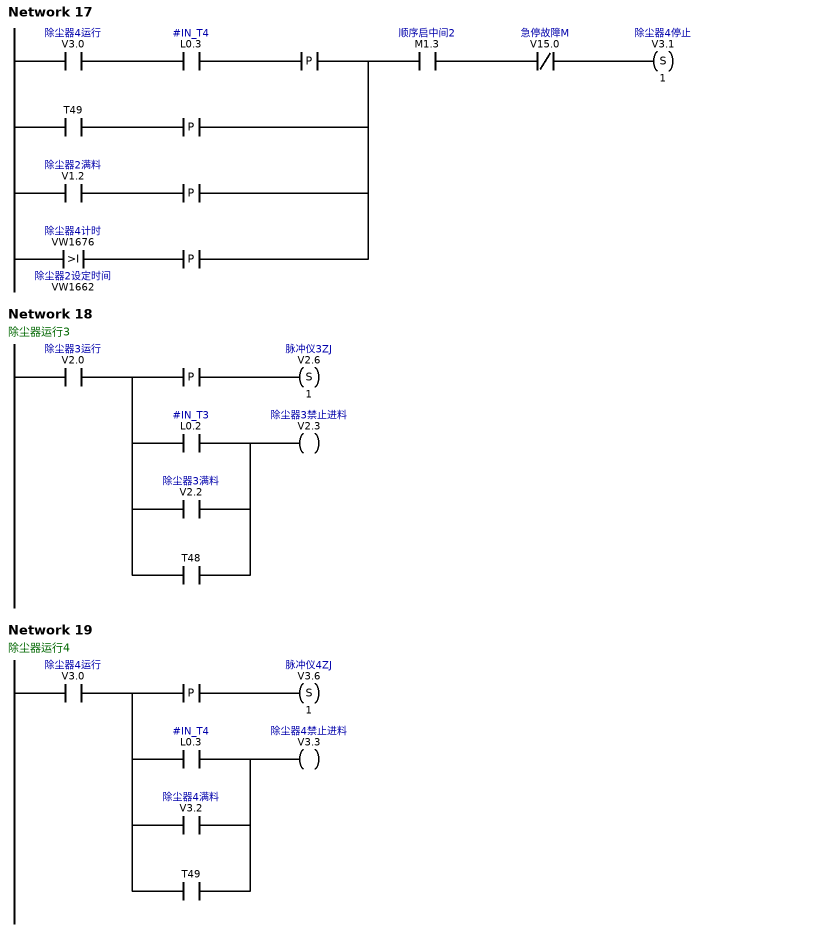
[picture p96: SBR29 networks 17-19]
Network 17
LD     除尘器4运行:V3.0
A      #IN_T4:L0.3
EU
LD     T49
EU
OLD
LD     除尘器2满料:V1.2
EU
OLD
LDW>   除尘器4计时:VW1676, 除尘器2设定时间:VW1662
EU
OLD
A      顺序启中间2:M1.3
AN     急停故障M:V15.0
S      除尘器4停止:V3.1, 1
Network 18
// 除尘器运行3
LD     除尘器3运行:V2.0
LPS
EU
S      脉冲仪3ZJ:V2.6, 1
LPP
LD     #IN_T3:L0.2
O      除尘器3满料:V2.2
O      T48
ALD
=      除尘器3禁止进料:V2.3
Network 19
// 除尘器运行4
LD     除尘器4运行:V3.0
LPS
EU
S      脉冲仪4ZJ:V3.6, 1
LPP
LD     #IN_T4:L0.3
O      除尘器4满料:V3.2
O      T49
ALD
=      除尘器4禁止进料:V3.3
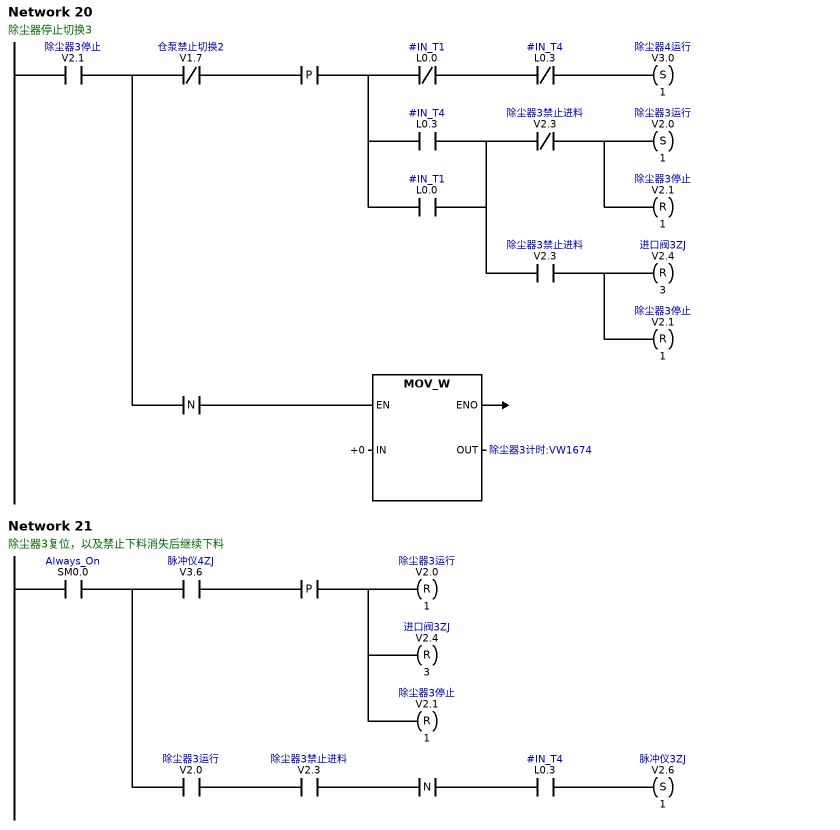
Network 20
// 除尘器停止切换3
LD     除尘器3停止:V2.1
LPS
AN     仓泵禁止切换2:V1.7
EU
LPS
AN     #IN_T1:L0.0
AN     #IN_T4:L0.3
S      除尘器4运行:V3.0, 1
LPP
LD     #IN_T4:L0.3
O      #IN_T1:L0.0
ALD
LPS
AN     除尘器3禁止进料:V2.3
S      除尘器3运行:V2.0, 1
R      除尘器3停止:V2.1, 1
LPP
A      除尘器3禁止进料:V2.3
R      进口阀3ZJ:V2.4, 3
R      除尘器3停止:V2.1, 1
LPP
ED
MOVW   +0, 除尘器3计时:VW1674
Network 21
// 除尘器3复位，以及禁止下料消失后继续下料
LD     Always_On:SM0.0
LPS
A      脉冲仪4ZJ:V3.6
EU
R      除尘器3运行:V2.0, 1
R      进口阀3ZJ:V2.4, 3
R      除尘器3停止:V2.1, 1
LPP
A      除尘器3运行:V2.0
A      除尘器3禁止进料:V2.3
ED
A      #IN_T4:L0.3
S      脉冲仪3ZJ:V2.6, 1
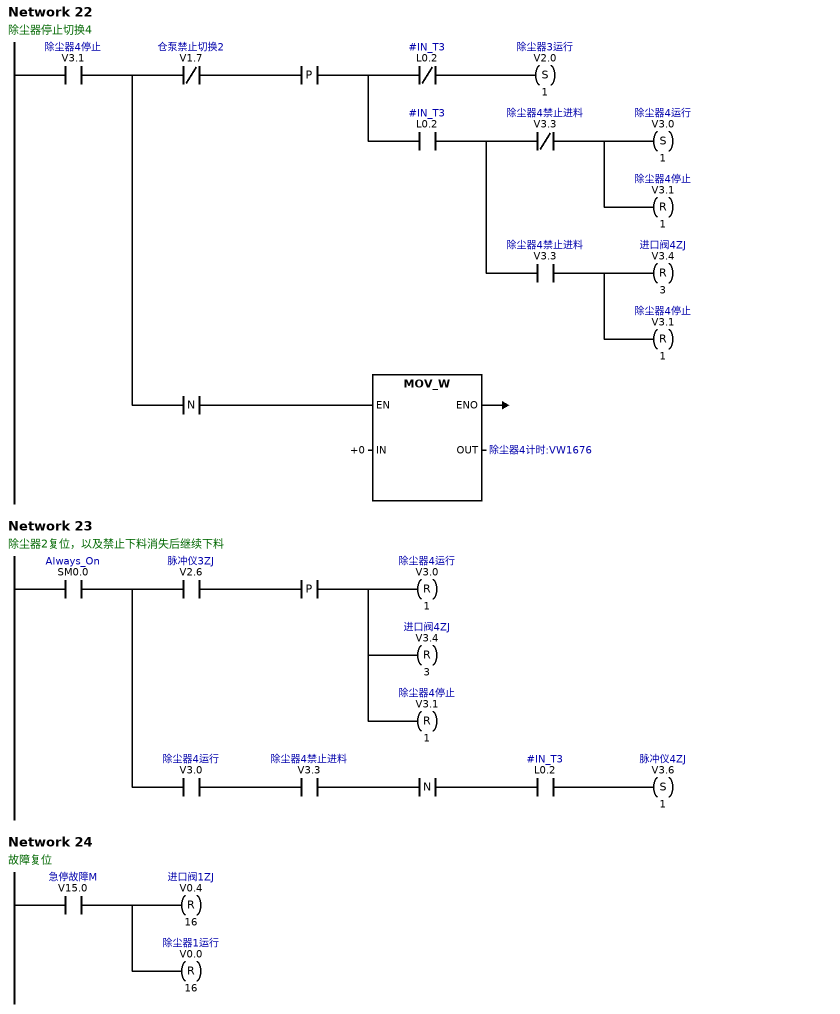
Network 22
// 除尘器停止切换4
LD     除尘器4停止:V3.1
LPS
AN     仓泵禁止切换2:V1.7
EU
LPS
AN     #IN_T3:L0.2
S      除尘器3运行:V2.0, 1
LPP
A      #IN_T3:L0.2
LPS
AN     除尘器4禁止进料:V3.3
S      除尘器4运行:V3.0, 1
R      除尘器4停止:V3.1, 1
LPP
A      除尘器4禁止进料:V3.3
R      进口阀4ZJ:V3.4, 3
R      除尘器4停止:V3.1, 1
LPP
ED
MOVW   +0, 除尘器4计时:VW1676
Network 23
// 除尘器2复位，以及禁止下料消失后继续下料
LD     Always_On:SM0.0
LPS
A      脉冲仪3ZJ:V2.6
EU
R      除尘器4运行:V3.0, 1
R      进口阀4ZJ:V3.4, 3
R      除尘器4停止:V3.1, 1
LPP
A      除尘器4运行:V3.0
A      除尘器4禁止进料:V3.3
ED
A      #IN_T3:L0.2
S      脉冲仪4ZJ:V3.6, 1
Network 24
// 故障复位
LD     急停故障M:V15.0
R      进口阀1ZJ:V0.4, 16
R      除尘器1运行:V0.0, 16
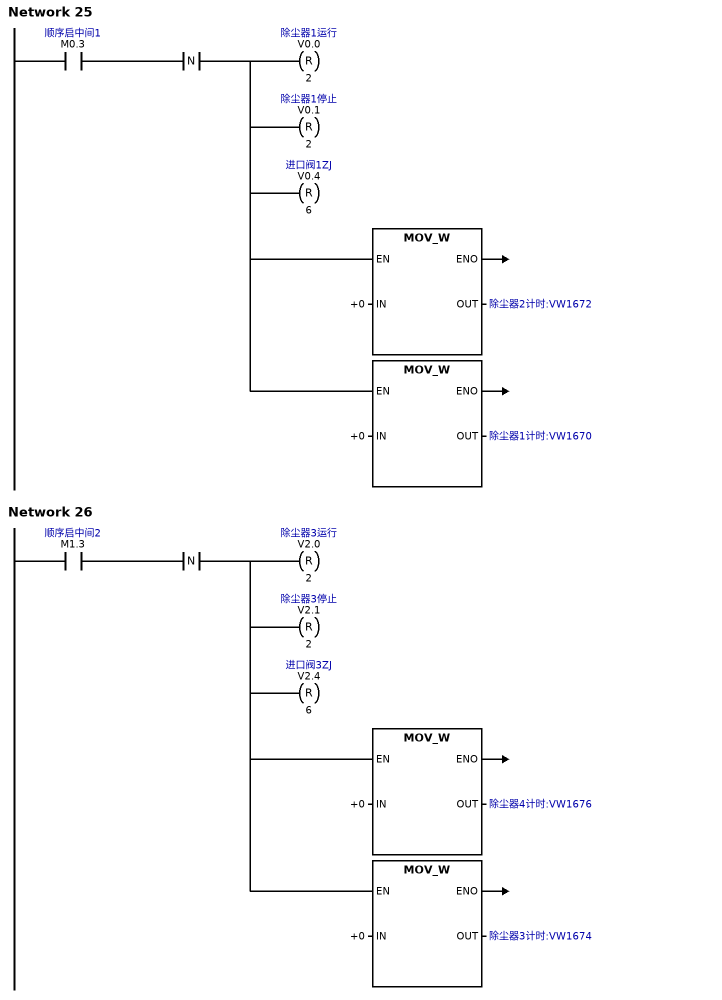
Network 25
LD     顺序启中间1:M0.3
ED
R      除尘器1运行:V0.0, 2
R      除尘器1停止:V0.1, 2
R      进口阀1ZJ:V0.4, 6
MOVW   +0, 除尘器2计时:VW1672
MOVW   +0, 除尘器1计时:VW1670
Network 26
LD     顺序启中间2:M1.3
ED
R      除尘器3运行:V2.0, 2
R      除尘器3停止:V2.1, 2
R      进口阀3ZJ:V2.4, 6
MOVW   +0, 除尘器4计时:VW1676
MOVW   +0, 除尘器3计时:VW1674
END_SUBROUTINE_BLOCK

SUBROUTINE_BLOCK MODBUS_XMZ:SBR50
TITLE=
BEGIN
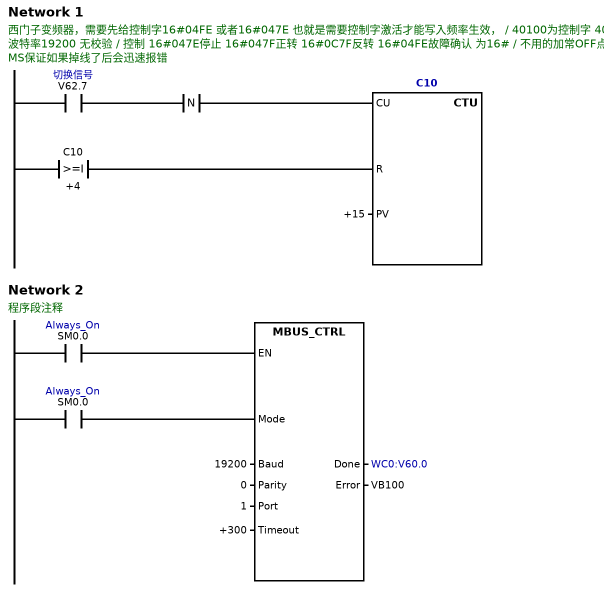
Network 1
// 西门子变频器，需要先给控制字16#04FE 或者16#047E 也就是需要控制字激活才能写入频率生效，
// 40100为控制字 40101为频率 0~16384=0~100% 
// 40342为频率 40345为电流 小数点通常2位  1  4
// 波特率19200 无校验
// 控制 16#047E停止 16#047F正转 16#0C7F反转 16#04FE故障确认 为16#
// 不用的加常OFF点屏蔽避免出错 也就是C10>=4时，=5的必须加常闭的sm0.0 超时300 MS保证如果掉线了后会迅速报错
LD     切换信号:V62.7
ED
LDW>=  C10, +4
CTU    C10, +15
Network 2
// 程序段注释
LD     Always_On:SM0.0
=      L60.0
LD     Always_On:SM0.0
=      L63.7
LD     L60.0
CALL   MBUS_CTRL:SBR2, L63.7, 19200, 0, 1, +300, WC0:V60.0, VB100
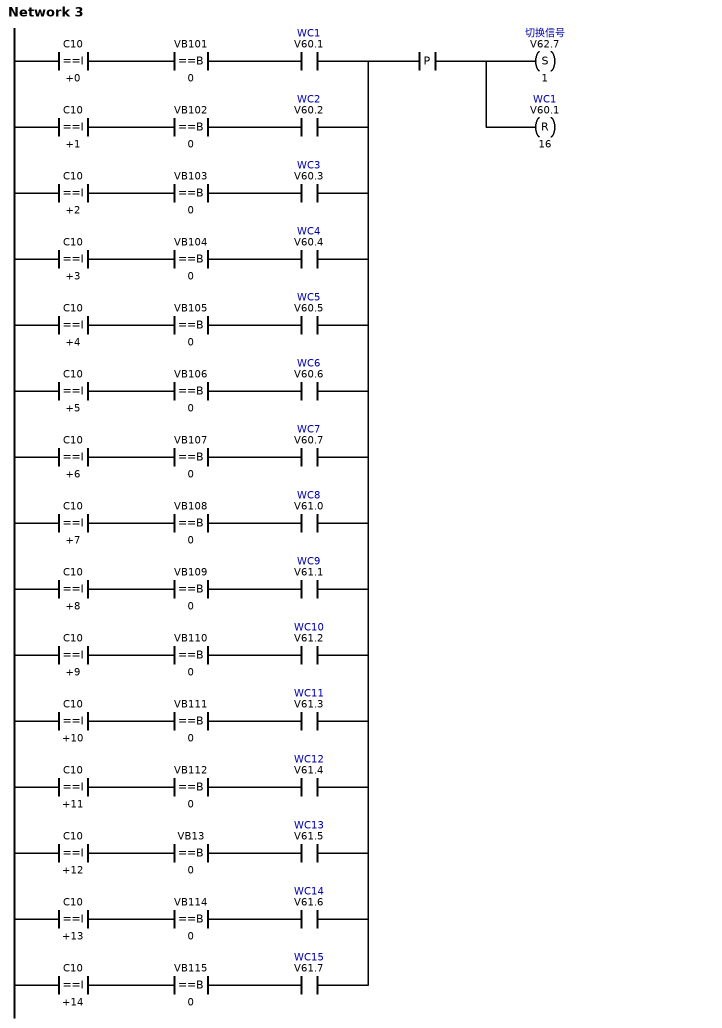
Network 3
LDW=   C10, +0
AB=    VB101, 0
A      WC1:V60.1
LDW=   C10, +1
AB=    VB102, 0
A      WC2:V60.2
OLD
LDW=   C10, +2
AB=    VB103, 0
A      WC3:V60.3
OLD
LDW=   C10, +3
AB=    VB104, 0
A      WC4:V60.4
OLD
LDW=   C10, +4
AB=    VB105, 0
A      WC5:V60.5
OLD
LDW=   C10, +5
AB=    VB106, 0
A      WC6:V60.6
OLD
LDW=   C10, +6
AB=    VB107, 0
A      WC7:V60.7
OLD
LDW=   C10, +7
AB=    VB108, 0
A      WC8:V61.0
OLD
LDW=   C10, +8
AB=    VB109, 0
A      WC9:V61.1
OLD
LDW=   C10, +9
AB=    VB110, 0
A      WC10:V61.2
OLD
LDW=   C10, +10
AB=    VB111, 0
A      WC11:V61.3
OLD
LDW=   C10, +11
AB=    VB112, 0
A      WC12:V61.4
OLD
LDW=   C10, +12
AB=    VB13, 0
A      WC13:V61.5
OLD
LDW=   C10, +13
AB=    VB114, 0
A      WC14:V61.6
OLD
LDW=   C10, +14
AB=    VB115, 0
A      WC15:V61.7
OLD
EU
S      切换信号:V62.7, 1
R      WC1:V60.1, 16
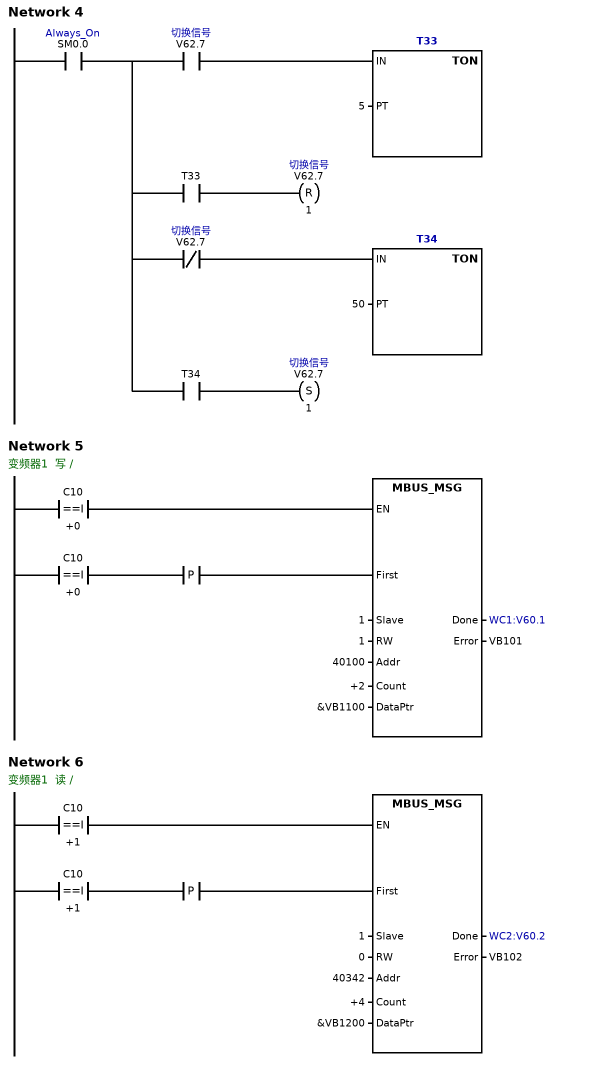
Network 4
LD     Always_On:SM0.0
LPS
A      切换信号:V62.7
TON    T33, 5
LRD
A      T33
R      切换信号:V62.7, 1
LRD
AN     切换信号:V62.7
TON    T34, 50
LPP
A      T34
S      切换信号:V62.7, 1
Network 5
// 变频器1  写
// 
LDW=   C10, +0
=      L60.0
LDW=   C10, +0
EU
=      L63.7
LD     L60.0
CALL   MBUS_MSG:SBR3, L63.7, 1, 1, 40100, +2, &VB1100, WC1:V60.1, VB101
Network 6
// 变频器1  读
// 
LDW=   C10, +1
=      L60.0
LDW=   C10, +1
EU
=      L63.7
LD     L60.0
CALL   MBUS_MSG:SBR3, L63.7, 1, 0, 40342, +4, &VB1200, WC2:V60.2, VB102
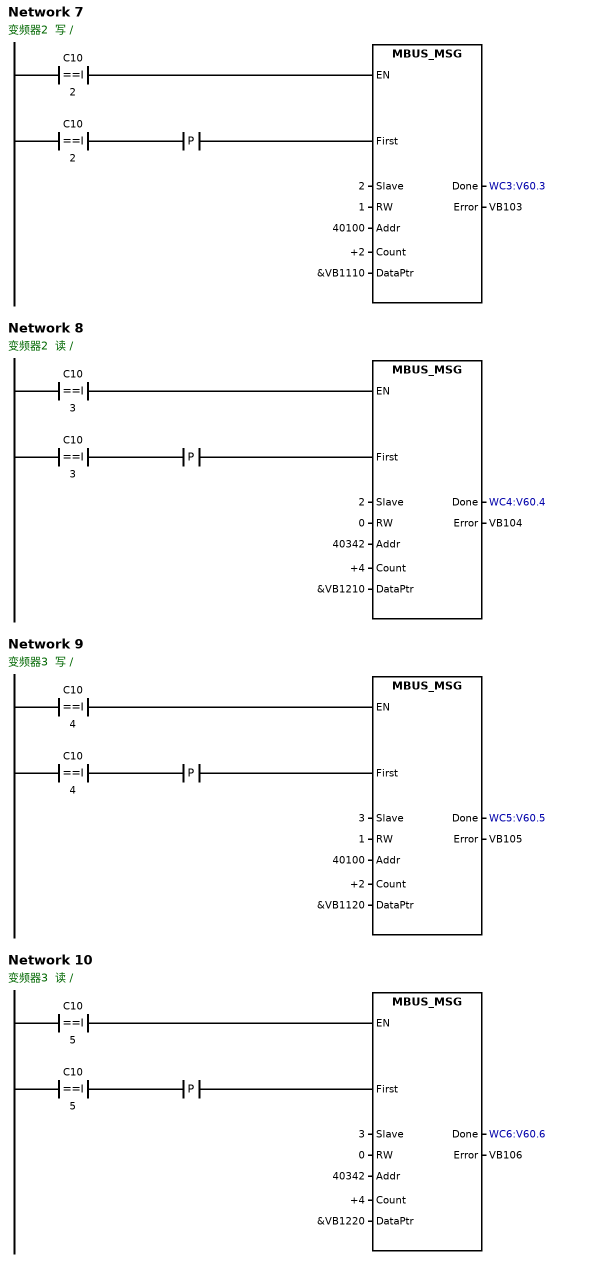
Network 7
// 变频器2  写
// 
LDW=   C10, 2
=      L60.0
LDW=   C10, 2
EU
=      L63.7
LD     L60.0
CALL   MBUS_MSG:SBR3, L63.7, 2, 1, 40100, +2, &VB1110, WC3:V60.3, VB103
Network 8
// 变频器2  读
// 
LDW=   C10, 3
=      L60.0
LDW=   C10, 3
EU
=      L63.7
LD     L60.0
CALL   MBUS_MSG:SBR3, L63.7, 2, 0, 40342, +4, &VB1210, WC4:V60.4, VB104
Network 9
// 变频器3  写
// 
LDW=   C10, 4
=      L60.0
LDW=   C10, 4
EU
=      L63.7
LD     L60.0
CALL   MBUS_MSG:SBR3, L63.7, 3, 1, 40100, +2, &VB1120, WC5:V60.5, VB105
Network 10
// 变频器3  读
// 
LDW=   C10, 5
=      L60.0
LDW=   C10, 5
EU
=      L63.7
LD     L60.0
CALL   MBUS_MSG:SBR3, L63.7, 3, 0, 40342, +4, &VB1220, WC6:V60.6, VB106
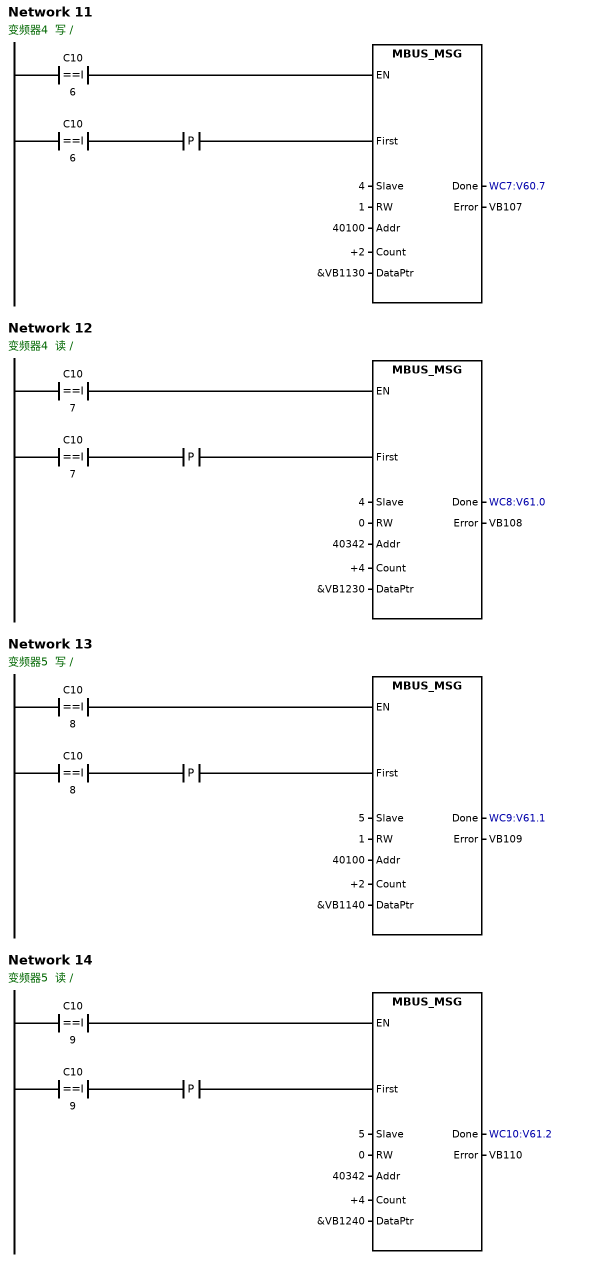
Network 11
// 变频器4  写
// 
LDW=   C10, 6
=      L60.0
LDW=   C10, 6
EU
=      L63.7
LD     L60.0
CALL   MBUS_MSG:SBR3, L63.7, 4, 1, 40100, +2, &VB1130, WC7:V60.7, VB107
Network 12
// 变频器4  读
// 
LDW=   C10, 7
=      L60.0
LDW=   C10, 7
EU
=      L63.7
LD     L60.0
CALL   MBUS_MSG:SBR3, L63.7, 4, 0, 40342, +4, &VB1230, WC8:V61.0, VB108
Network 13
// 变频器5  写
// 
LDW=   C10, 8
=      L60.0
LDW=   C10, 8
EU
=      L63.7
LD     L60.0
CALL   MBUS_MSG:SBR3, L63.7, 5, 1, 40100, +2, &VB1140, WC9:V61.1, VB109
Network 14
// 变频器5  读
// 
LDW=   C10, 9
=      L60.0
LDW=   C10, 9
EU
=      L63.7
LD     L60.0
CALL   MBUS_MSG:SBR3, L63.7, 5, 0, 40342, +4, &VB1240, WC10:V61.2, VB110
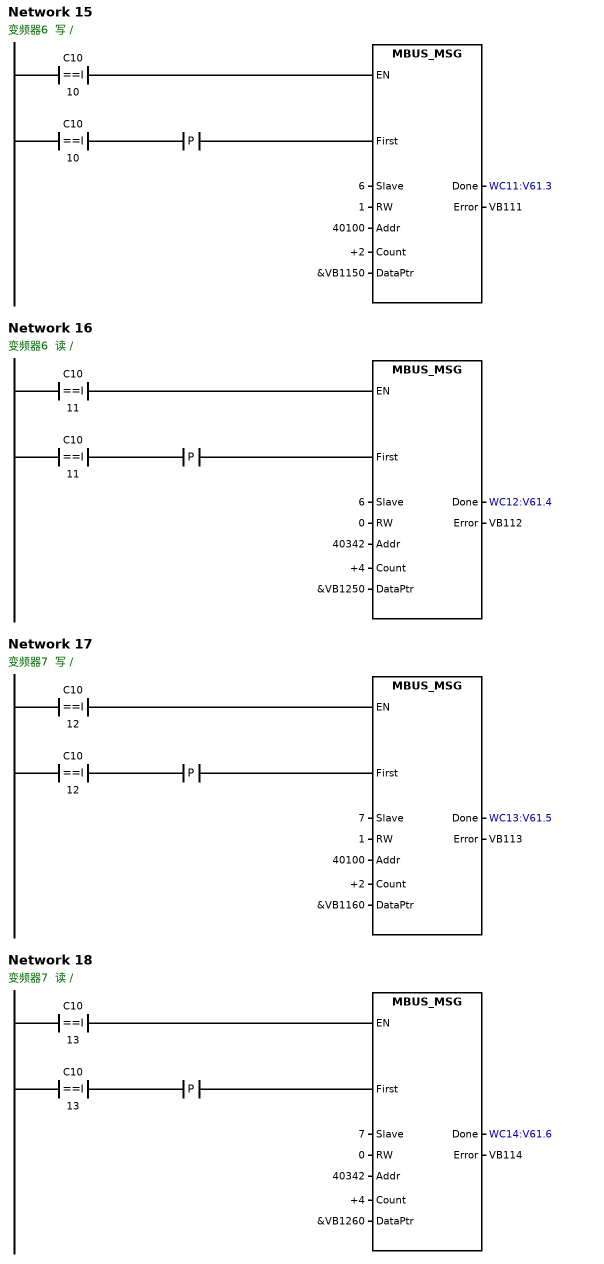
Network 15
// 变频器6  写
// 
LDW=   C10, 10
=      L60.0
LDW=   C10, 10
EU
=      L63.7
LD     L60.0
CALL   MBUS_MSG:SBR3, L63.7, 6, 1, 40100, +2, &VB1150, WC11:V61.3, VB111
Network 16
// 变频器6  读
// 
LDW=   C10, 11
=      L60.0
LDW=   C10, 11
EU
=      L63.7
LD     L60.0
CALL   MBUS_MSG:SBR3, L63.7, 6, 0, 40342, +4, &VB1250, WC12:V61.4, VB112
Network 17
// 变频器7  写
// 
LDW=   C10, 12
=      L60.0
LDW=   C10, 12
EU
=      L63.7
LD     L60.0
CALL   MBUS_MSG:SBR3, L63.7, 7, 1, 40100, +2, &VB1160, WC13:V61.5, VB113
Network 18
// 变频器7  读
// 
LDW=   C10, 13
=      L60.0
LDW=   C10, 13
EU
=      L63.7
LD     L60.0
CALL   MBUS_MSG:SBR3, L63.7, 7, 0, 40342, +4, &VB1260, WC14:V61.6, VB114
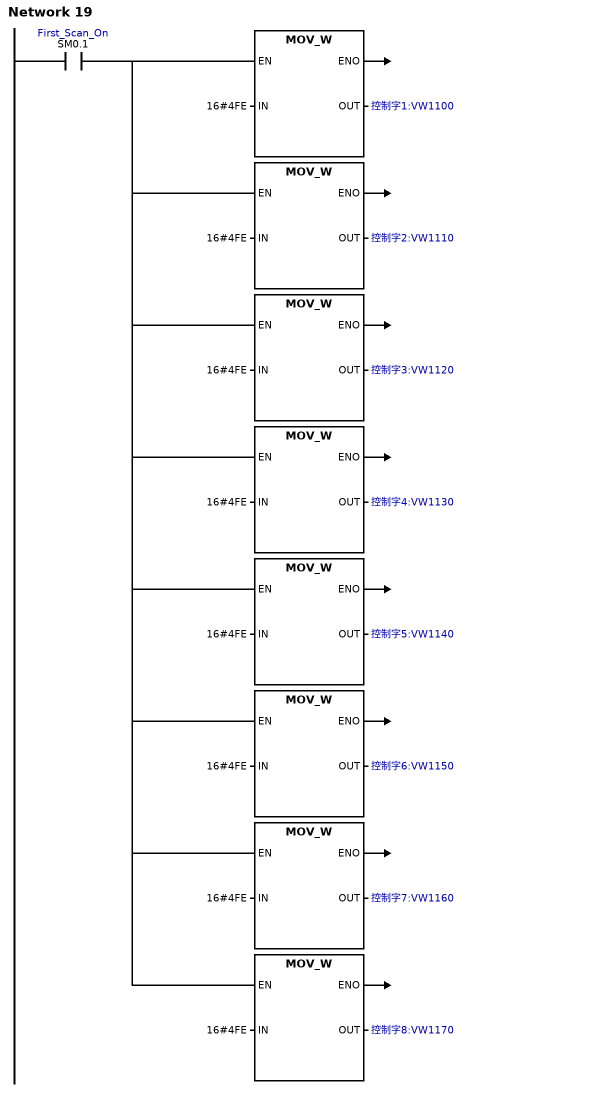
Network 19
LD     First_Scan_On:SM0.1
MOVW   16#4FE, 控制字1:VW1100
MOVW   16#4FE, 控制字2:VW1110
MOVW   16#4FE, 控制字3:VW1120
MOVW   16#4FE, 控制字4:VW1130
MOVW   16#4FE, 控制字5:VW1140
MOVW   16#4FE, 控制字6:VW1150
MOVW   16#4FE, 控制字7:VW1160
MOVW   16#4FE, 控制字8:VW1170
END_SUBROUTINE_BLOCK

SUBROUTINE_BLOCK MODBUS_SND:SBR51
TITLE=
BEGIN
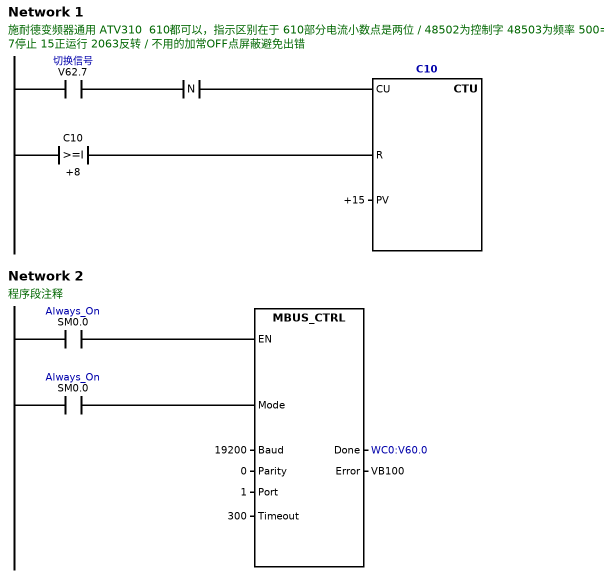
Network 1
// 施耐德变频器通用 ATV310  610都可以，指示区别在于 610部分电流小数点是两位
// 48502为控制字 48503为频率 500=50.0HZ
// 43202为状态字 43203为频率  43205为电流  2 4
// 波特率19200 无校验
// 控制字 6准备 7停止 15正运行 2063反转
// 不用的加常OFF点屏蔽避免出错
LD     切换信号:V62.7
ED
LDW>=  C10, +8
CTU    C10, +15
Network 2
// 程序段注释
LD     Always_On:SM0.0
=      L60.0
LD     Always_On:SM0.0
=      L63.7
LD     L60.0
CALL   MBUS_CTRL:SBR2, L63.7, 19200, 0, 1, 300, WC0:V60.0, VB100
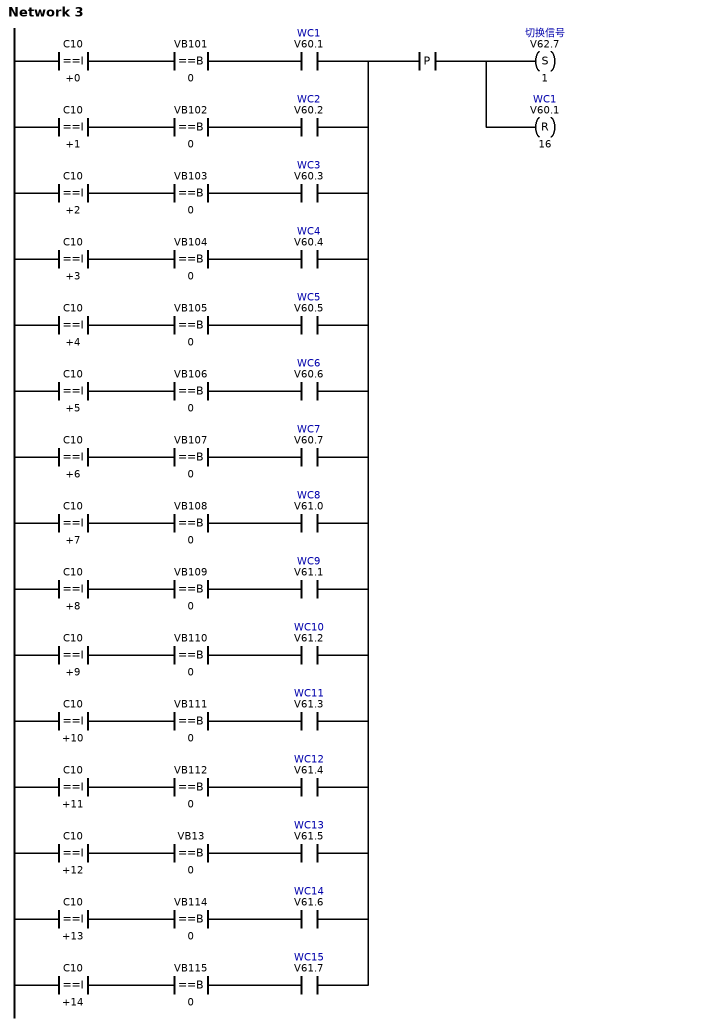
Network 3
LDW=   C10, +0
AB=    VB101, 0
A      WC1:V60.1
LDW=   C10, +1
AB=    VB102, 0
A      WC2:V60.2
OLD
LDW=   C10, +2
AB=    VB103, 0
A      WC3:V60.3
OLD
LDW=   C10, +3
AB=    VB104, 0
A      WC4:V60.4
OLD
LDW=   C10, +4
AB=    VB105, 0
A      WC5:V60.5
OLD
LDW=   C10, +5
AB=    VB106, 0
A      WC6:V60.6
OLD
LDW=   C10, +6
AB=    VB107, 0
A      WC7:V60.7
OLD
LDW=   C10, +7
AB=    VB108, 0
A      WC8:V61.0
OLD
LDW=   C10, +8
AB=    VB109, 0
A      WC9:V61.1
OLD
LDW=   C10, +9
AB=    VB110, 0
A      WC10:V61.2
OLD
LDW=   C10, +10
AB=    VB111, 0
A      WC11:V61.3
OLD
LDW=   C10, +11
AB=    VB112, 0
A      WC12:V61.4
OLD
LDW=   C10, +12
AB=    VB13, 0
A      WC13:V61.5
OLD
LDW=   C10, +13
AB=    VB114, 0
A      WC14:V61.6
OLD
LDW=   C10, +14
AB=    VB115, 0
A      WC15:V61.7
OLD
EU
S      切换信号:V62.7, 1
R      WC1:V60.1, 16
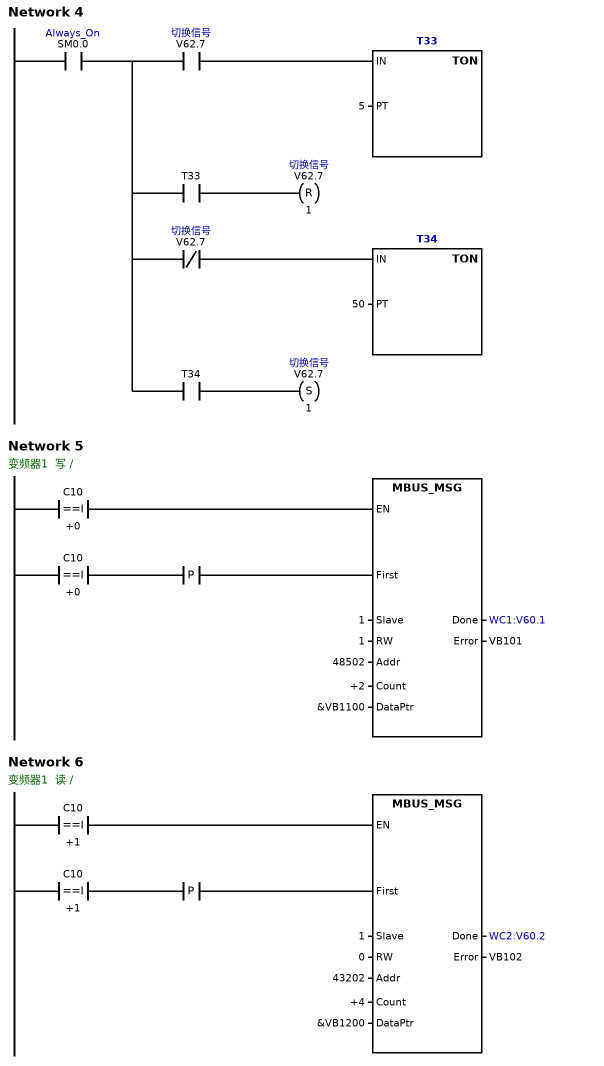
Network 4
LD     Always_On:SM0.0
LPS
A      切换信号:V62.7
TON    T33, 5
LRD
A      T33
R      切换信号:V62.7, 1
LRD
AN     切换信号:V62.7
TON    T34, 50
LPP
A      T34
S      切换信号:V62.7, 1
Network 5
// 变频器1  写
// 
LDW=   C10, +0
=      L60.0
LDW=   C10, +0
EU
=      L63.7
LD     L60.0
CALL   MBUS_MSG:SBR3, L63.7, 1, 1, 48502, +2, &VB1100, WC1:V60.1, VB101
Network 6
// 变频器1  读
// 
LDW=   C10, +1
=      L60.0
LDW=   C10, +1
EU
=      L63.7
LD     L60.0
CALL   MBUS_MSG:SBR3, L63.7, 1, 0, 43202, +4, &VB1200, WC2:V60.2, VB102
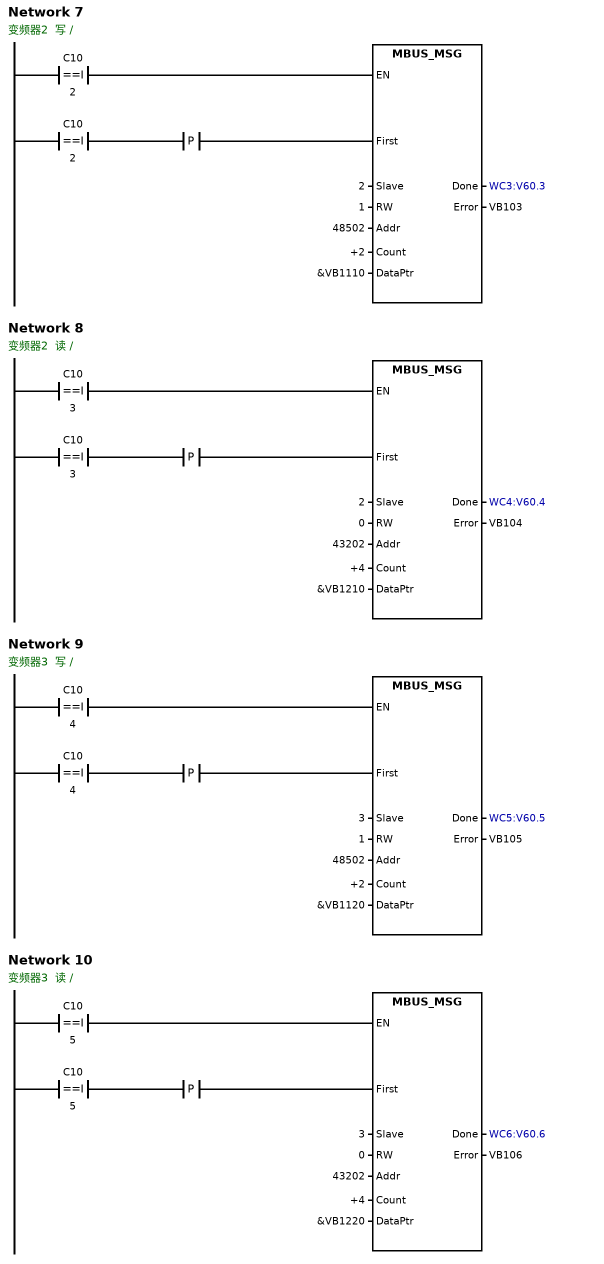
Network 7
// 变频器2  写
// 
LDW=   C10, 2
=      L60.0
LDW=   C10, 2
EU
=      L63.7
LD     L60.0
CALL   MBUS_MSG:SBR3, L63.7, 2, 1, 48502, +2, &VB1110, WC3:V60.3, VB103
Network 8
// 变频器2  读
// 
LDW=   C10, 3
=      L60.0
LDW=   C10, 3
EU
=      L63.7
LD     L60.0
CALL   MBUS_MSG:SBR3, L63.7, 2, 0, 43202, +4, &VB1210, WC4:V60.4, VB104
Network 9
// 变频器3  写
// 
LDW=   C10, 4
=      L60.0
LDW=   C10, 4
EU
=      L63.7
LD     L60.0
CALL   MBUS_MSG:SBR3, L63.7, 3, 1, 48502, +2, &VB1120, WC5:V60.5, VB105
Network 10
// 变频器3  读
// 
LDW=   C10, 5
=      L60.0
LDW=   C10, 5
EU
=      L63.7
LD     L60.0
CALL   MBUS_MSG:SBR3, L63.7, 3, 0, 43202, +4, &VB1220, WC6:V60.6, VB106
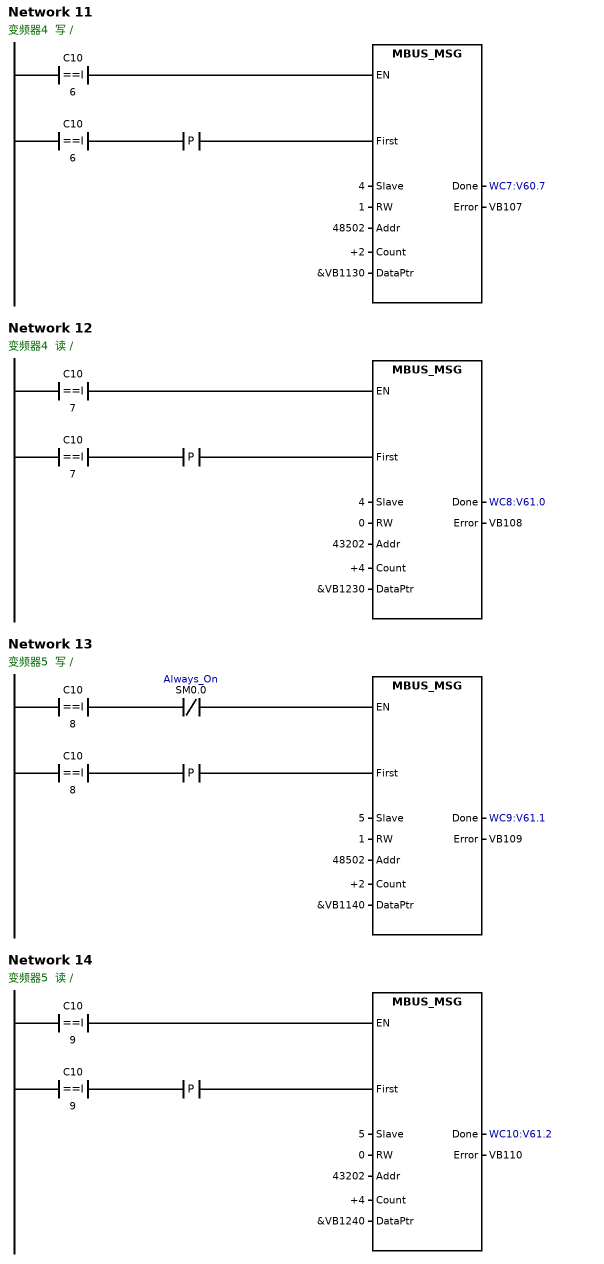
Network 11
// 变频器4  写
// 
LDW=   C10, 6
=      L60.0
LDW=   C10, 6
EU
=      L63.7
LD     L60.0
CALL   MBUS_MSG:SBR3, L63.7, 4, 1, 48502, +2, &VB1130, WC7:V60.7, VB107
Network 12
// 变频器4  读
// 
LDW=   C10, 7
=      L60.0
LDW=   C10, 7
EU
=      L63.7
LD     L60.0
CALL   MBUS_MSG:SBR3, L63.7, 4, 0, 43202, +4, &VB1230, WC8:V61.0, VB108
Network 13
// 变频器5  写
// 
LDW=   C10, 8
AN     Always_On:SM0.0
=      L60.0
LDW=   C10, 8
EU
=      L63.7
LD     L60.0
CALL   MBUS_MSG:SBR3, L63.7, 5, 1, 48502, +2, &VB1140, WC9:V61.1, VB109
Network 14
// 变频器5  读
// 
LDW=   C10, 9
=      L60.0
LDW=   C10, 9
EU
=      L63.7
LD     L60.0
CALL   MBUS_MSG:SBR3, L63.7, 5, 0, 43202, +4, &VB1240, WC10:V61.2, VB110
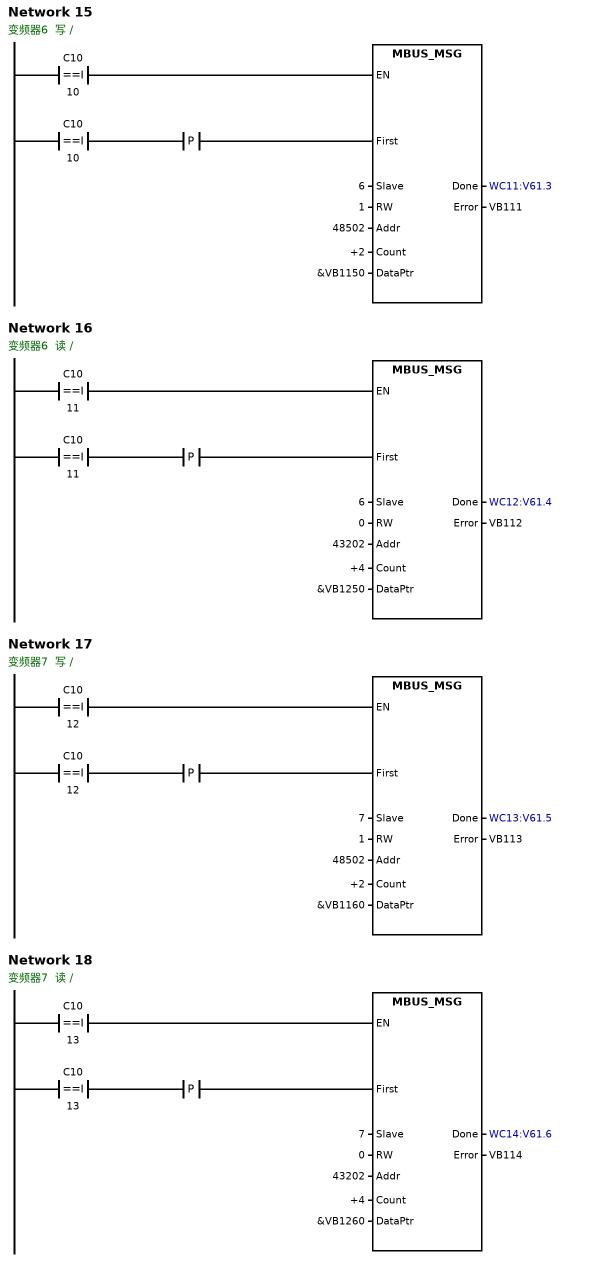
Network 15
// 变频器6  写
// 
LDW=   C10, 10
=      L60.0
LDW=   C10, 10
EU
=      L63.7
LD     L60.0
CALL   MBUS_MSG:SBR3, L63.7, 6, 1, 48502, +2, &VB1150, WC11:V61.3, VB111
Network 16
// 变频器6  读
// 
LDW=   C10, 11
=      L60.0
LDW=   C10, 11
EU
=      L63.7
LD     L60.0
CALL   MBUS_MSG:SBR3, L63.7, 6, 0, 43202, +4, &VB1250, WC12:V61.4, VB112
Network 17
// 变频器7  写
// 
LDW=   C10, 12
=      L60.0
LDW=   C10, 12
EU
=      L63.7
LD     L60.0
CALL   MBUS_MSG:SBR3, L63.7, 7, 1, 48502, +2, &VB1160, WC13:V61.5, VB113
Network 18
// 变频器7  读
// 
LDW=   C10, 13
=      L60.0
LDW=   C10, 13
EU
=      L63.7
LD     L60.0
CALL   MBUS_MSG:SBR3, L63.7, 7, 0, 43202, +4, &VB1260, WC14:V61.6, VB114
END_SUBROUTINE_BLOCK

SUBROUTINE_BLOCK MODBUS_TD:SBR52
TITLE=
BEGIN
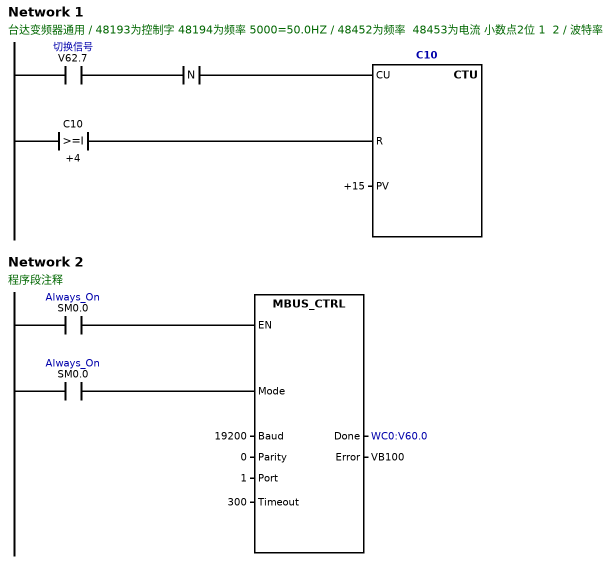
Network 1
// 台达变频器通用
// 48193为控制字 48194为频率 5000=50.0HZ
// 48452为频率  48453为电流 小数点2位 1  2
// 波特率19200 无校验
// 不用的加常OFF点屏蔽避免出错
LD     切换信号:V62.7
ED
LDW>=  C10, +4
CTU    C10, +15
Network 2
// 程序段注释
LD     Always_On:SM0.0
=      L60.0
LD     Always_On:SM0.0
=      L63.7
LD     L60.0
CALL   MBUS_CTRL:SBR2, L63.7, 19200, 0, 1, 300, WC0:V60.0, VB100
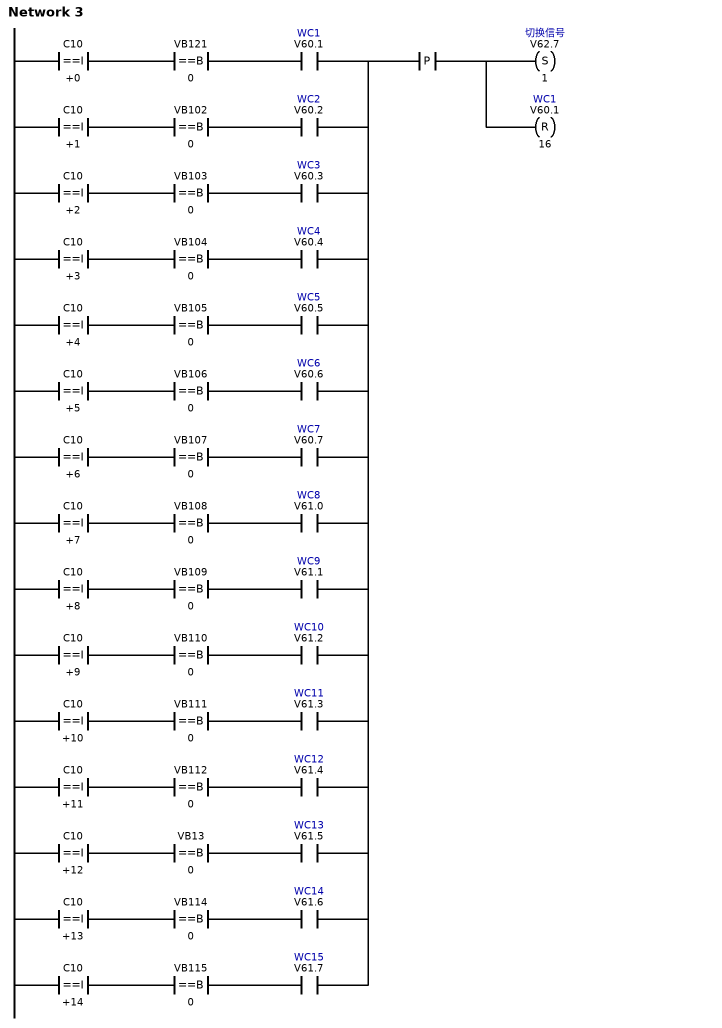
Network 3
LDW=   C10, +0
AB=    VB121, 0
A      WC1:V60.1
LDW=   C10, +1
AB=    VB102, 0
A      WC2:V60.2
OLD
LDW=   C10, +2
AB=    VB103, 0
A      WC3:V60.3
OLD
LDW=   C10, +3
AB=    VB104, 0
A      WC4:V60.4
OLD
LDW=   C10, +4
AB=    VB105, 0
A      WC5:V60.5
OLD
LDW=   C10, +5
AB=    VB106, 0
A      WC6:V60.6
OLD
LDW=   C10, +6
AB=    VB107, 0
A      WC7:V60.7
OLD
LDW=   C10, +7
AB=    VB108, 0
A      WC8:V61.0
OLD
LDW=   C10, +8
AB=    VB109, 0
A      WC9:V61.1
OLD
LDW=   C10, +9
AB=    VB110, 0
A      WC10:V61.2
OLD
LDW=   C10, +10
AB=    VB111, 0
A      WC11:V61.3
OLD
LDW=   C10, +11
AB=    VB112, 0
A      WC12:V61.4
OLD
LDW=   C10, +12
AB=    VB13, 0
A      WC13:V61.5
OLD
LDW=   C10, +13
AB=    VB114, 0
A      WC14:V61.6
OLD
LDW=   C10, +14
AB=    VB115, 0
A      WC15:V61.7
OLD
EU
S      切换信号:V62.7, 1
R      WC1:V60.1, 16
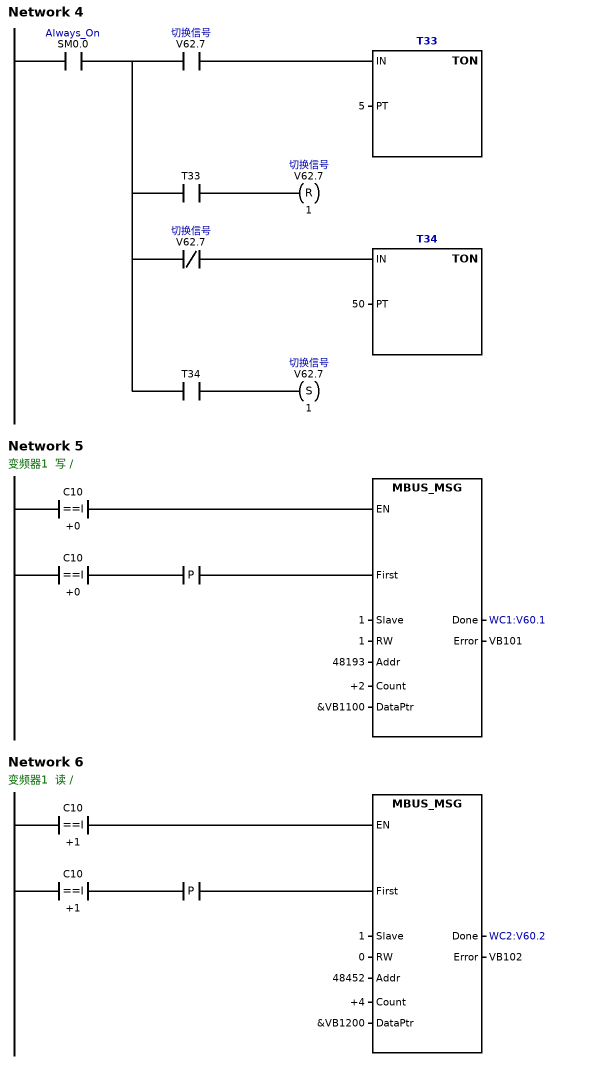
Network 4
LD     Always_On:SM0.0
LPS
A      切换信号:V62.7
TON    T33, 5
LRD
A      T33
R      切换信号:V62.7, 1
LRD
AN     切换信号:V62.7
TON    T34, 50
LPP
A      T34
S      切换信号:V62.7, 1
Network 5
// 变频器1  写
// 
LDW=   C10, +0
=      L60.0
LDW=   C10, +0
EU
=      L63.7
LD     L60.0
CALL   MBUS_MSG:SBR3, L63.7, 1, 1, 48193, +2, &VB1100, WC1:V60.1, VB101
Network 6
// 变频器1  读
// 
LDW=   C10, +1
=      L60.0
LDW=   C10, +1
EU
=      L63.7
LD     L60.0
CALL   MBUS_MSG:SBR3, L63.7, 1, 0, 48452, +4, &VB1200, WC2:V60.2, VB102
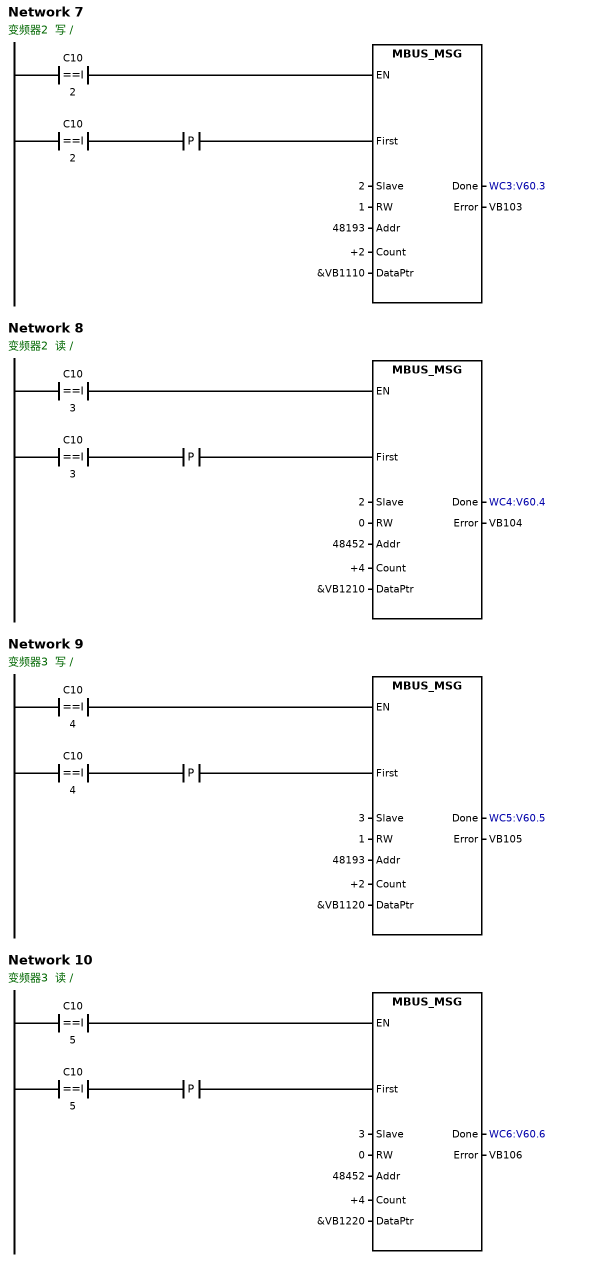
Network 7
// 变频器2  写
// 
LDW=   C10, 2
=      L60.0
LDW=   C10, 2
EU
=      L63.7
LD     L60.0
CALL   MBUS_MSG:SBR3, L63.7, 2, 1, 48193, +2, &VB1110, WC3:V60.3, VB103
Network 8
// 变频器2  读
// 
LDW=   C10, 3
=      L60.0
LDW=   C10, 3
EU
=      L63.7
LD     L60.0
CALL   MBUS_MSG:SBR3, L63.7, 2, 0, 48452, +4, &VB1210, WC4:V60.4, VB104
Network 9
// 变频器3  写
// 
LDW=   C10, 4
=      L60.0
LDW=   C10, 4
EU
=      L63.7
LD     L60.0
CALL   MBUS_MSG:SBR3, L63.7, 3, 1, 48193, +2, &VB1120, WC5:V60.5, VB105
Network 10
// 变频器3  读
// 
LDW=   C10, 5
=      L60.0
LDW=   C10, 5
EU
=      L63.7
LD     L60.0
CALL   MBUS_MSG:SBR3, L63.7, 3, 0, 48452, +4, &VB1220, WC6:V60.6, VB106
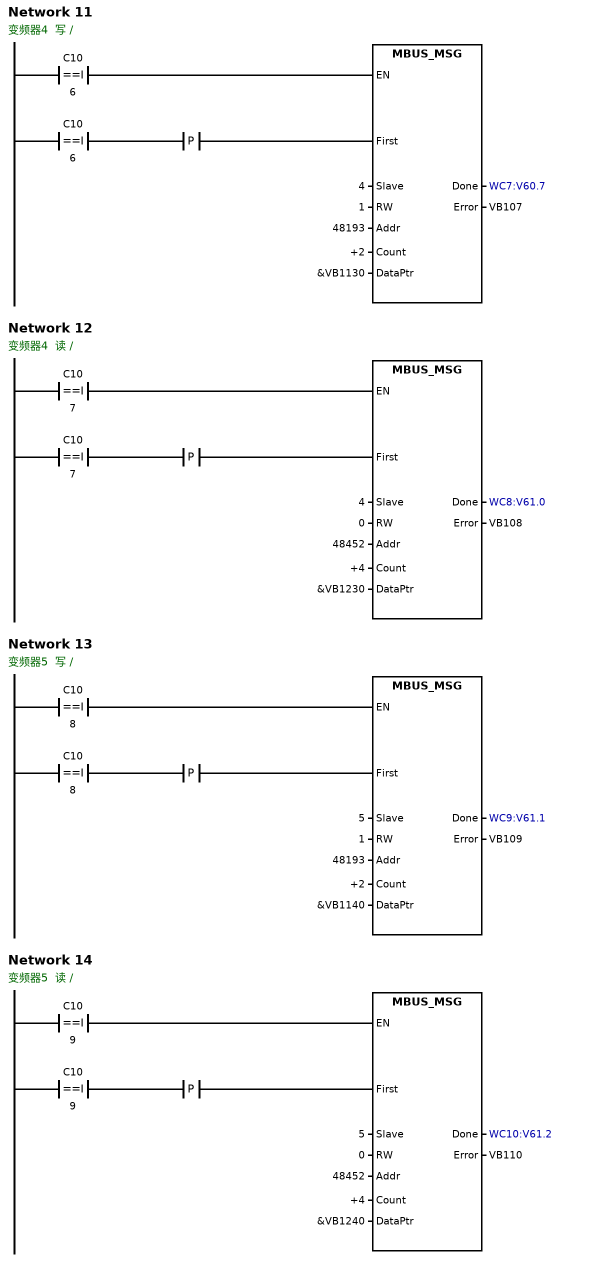
Network 11
// 变频器4  写
// 
LDW=   C10, 6
=      L60.0
LDW=   C10, 6
EU
=      L63.7
LD     L60.0
CALL   MBUS_MSG:SBR3, L63.7, 4, 1, 48193, +2, &VB1130, WC7:V60.7, VB107
Network 12
// 变频器4  读
// 
LDW=   C10, 7
=      L60.0
LDW=   C10, 7
EU
=      L63.7
LD     L60.0
CALL   MBUS_MSG:SBR3, L63.7, 4, 0, 48452, +4, &VB1230, WC8:V61.0, VB108
Network 13
// 变频器5  写
// 
LDW=   C10, 8
=      L60.0
LDW=   C10, 8
EU
=      L63.7
LD     L60.0
CALL   MBUS_MSG:SBR3, L63.7, 5, 1, 48193, +2, &VB1140, WC9:V61.1, VB109
Network 14
// 变频器5  读
// 
LDW=   C10, 9
=      L60.0
LDW=   C10, 9
EU
=      L63.7
LD     L60.0
CALL   MBUS_MSG:SBR3, L63.7, 5, 0, 48452, +4, &VB1240, WC10:V61.2, VB110
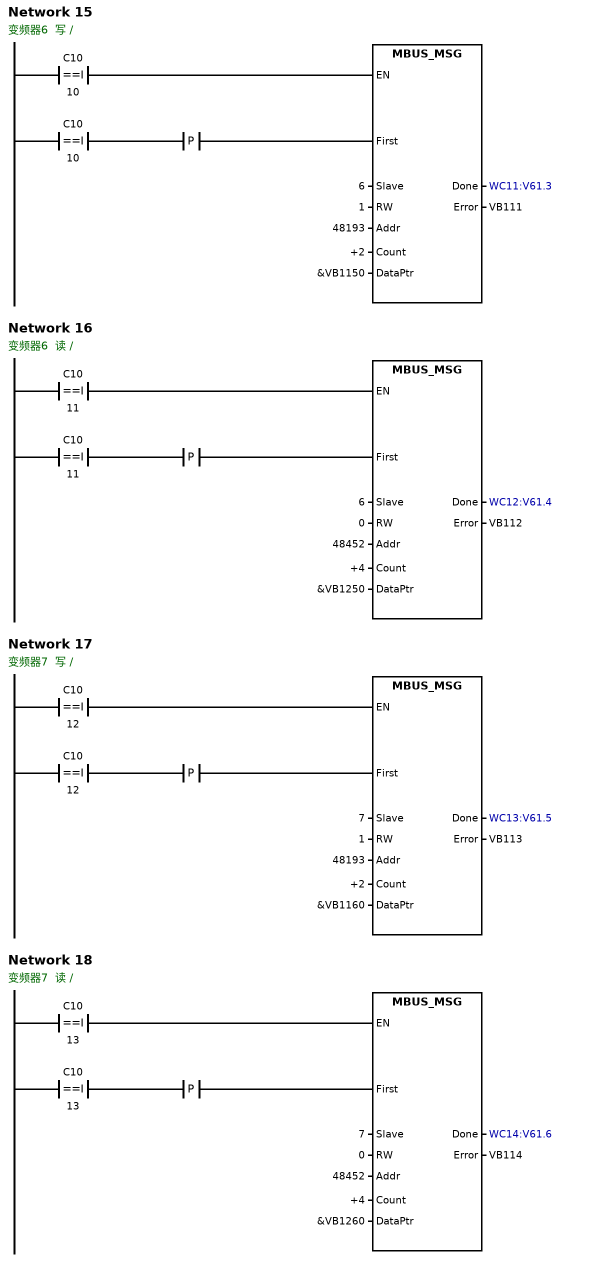
Network 15
// 变频器6  写
// 
LDW=   C10, 10
=      L60.0
LDW=   C10, 10
EU
=      L63.7
LD     L60.0
CALL   MBUS_MSG:SBR3, L63.7, 6, 1, 48193, +2, &VB1150, WC11:V61.3, VB111
Network 16
// 变频器6  读
// 
LDW=   C10, 11
=      L60.0
LDW=   C10, 11
EU
=      L63.7
LD     L60.0
CALL   MBUS_MSG:SBR3, L63.7, 6, 0, 48452, +4, &VB1250, WC12:V61.4, VB112
Network 17
// 变频器7  写
// 
LDW=   C10, 12
=      L60.0
LDW=   C10, 12
EU
=      L63.7
LD     L60.0
CALL   MBUS_MSG:SBR3, L63.7, 7, 1, 48193, +2, &VB1160, WC13:V61.5, VB113
Network 18
// 变频器7  读
// 
LDW=   C10, 13
=      L60.0
LDW=   C10, 13
EU
=      L63.7
LD     L60.0
CALL   MBUS_MSG:SBR3, L63.7, 7, 0, 48452, +4, &VB1260, WC14:V61.6, VB114
END_SUBROUTINE_BLOCK

SUBROUTINE_BLOCK MODBUS_AT:SBR53
TITLE=
BEGIN
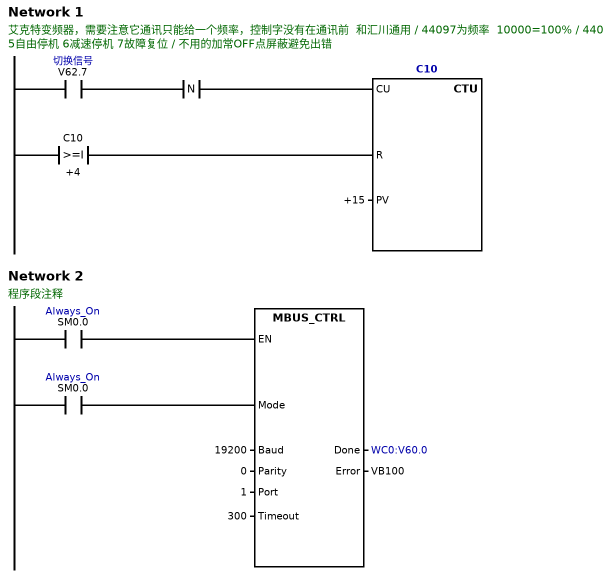
Network 1
// 艾克特变频器，需要注意它通讯只能给一个频率，控制字没有在通讯前  和汇川通用
// 44097为频率  10000=100%
// 44098为频率 44101为电流  通常为2位小数点  1  4
// 波特率19200 无校验
// 48193 控制 1正转 2反转 5自由停机 6减速停机 7故障复位
// 不用的加常OFF点屏蔽避免出错
LD     切换信号:V62.7
ED
LDW>=  C10, +4
CTU    C10, +15
Network 2
// 程序段注释
LD     Always_On:SM0.0
=      L60.0
LD     Always_On:SM0.0
=      L63.7
LD     L60.0
CALL   MBUS_CTRL:SBR2, L63.7, 19200, 0, 1, 300, WC0:V60.0, VB100
